(* PLC project Unbenannt, Unbekannt Unbenannt 1 *)
(* stored: creationDateTime 2019-09-13T11:08:45, modificationDateTime 2019-09-13T11:39:11 *)

PROGRAM program0
  VAR
    LocalVar0 : DINT;
    LocalVar1 : DINT;
    LocalVar2 : DINT;
  END_VAR

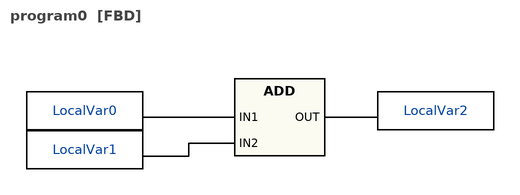
(* FBD diagram, written out as Structured Text *)
LocalVar2 := LocalVar0 + LocalVar1;
END_PROGRAM

(* this function will initialize a given array of byte with 0 *)
FUNCTION_BLOCK _BUFFER_CLEAR
  VAR_INPUT
    SIZE : UINT;
  END_VAR
  VAR_OUTPUT
    BUFFER_CLEAR : BOOL;
  END_VAR
  VAR_IN_OUT
    PT : ARRAY[0..249] OF BYTE;
  END_VAR
  VAR
    err : INT;
    result : WORD;
  END_VAR

            result:=MEMSET(err,BYTE#00,UINT_TO_DINT(size),pt[0]);

BUFFER_CLEAR := (err = 0);




          
END_FUNCTION_BLOCK

CONFIGURATION Config0
  RESOURCE Res0 ON PLC
    TASK task0(INTERVAL := T#20ms, PRIORITY := 0);
    PROGRAM instance0 WITH task0 : program0;
  END_RESOURCE
END_CONFIGURATION
